// LS Electric XG5000 project: 1129_PLC_Simulator_LS
// PLC NewPLC
// module base 0 slot 0: 입출력 모듈:XBC-DR20S (DC 24V 입력 12점, 릴레이 출력 8점)

PROGRAM simulator_test (task: 스캔 프로그램)

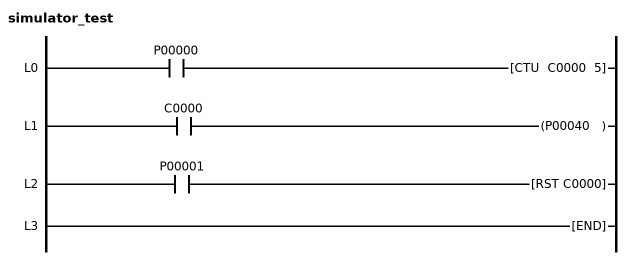
; L0
LOAD      P00000
CTU       C0000 5
; L1
LOAD      C0000
OUT       P00040
; L2
LOAD      P00001
RST       C0000
; L3
END